{attribute 'qualified_only'}
VAR_GLOBAL
	bSimulatorOn : BOOL;
	fPistonSidePressure : LREAL;
	fRodSidePressure 	: LREAL;
	fPistonPosition 	: LREAL;
END_VAR

(* stored: Version 1.1.0.1, ProductVersion 3.1.4024.10
   GVL G_Simulator: Id {7f848778-065f-4410-a7b4-047e2d0f684b} *)
